// SIMATIC S7-200 project (STEP 7-Micro/WIN), CPU 224XP REL 02.01

SYMBOL_TABLE USER1
send_enable      V1020.0
gps_lat_deg      VW50
gps_lat_min      VD52
gps_lat_dir      VB56
gps_long_deg     VW57
gps_long_min     VD59
gps_long_dir     VB64
gps_alt          VD65
gps_alt_u        VB69
gps_speed        VD70
msg              VB2000
counter          VW100
counter_delay    VW102
counter_send     V10.0
counter_max      VW104
counter_stop     V10.1
table            VW2500
table_count      VW2502
table_out        VW110
table_out_s      VB112
init_pin         VB1001
init_srv         VB1006
init_busy        V1000.0
init_done        V1000.1
init_ab          V1000.2
init_st          VW1026
send_ready       V1100.3
send_to          VB1050
send_busy        V1100.0
send_done        V1100.1
send_ab          V1100.2
send_st          VW1126
send_en          V1100.4
send_stop        V1100.5
rcv_busy         V1200.0
rcv_done         V1200.1
rcv_ab           V1200.2
rcv_buf          VB1210
rcv_msg          VB1238
rcv_st           VW1250
END_SYMBOL_TABLE

ORGANIZATION_BLOCK MAIN:OB1
TITLE=PROGRAM COMMENTS
BEGIN
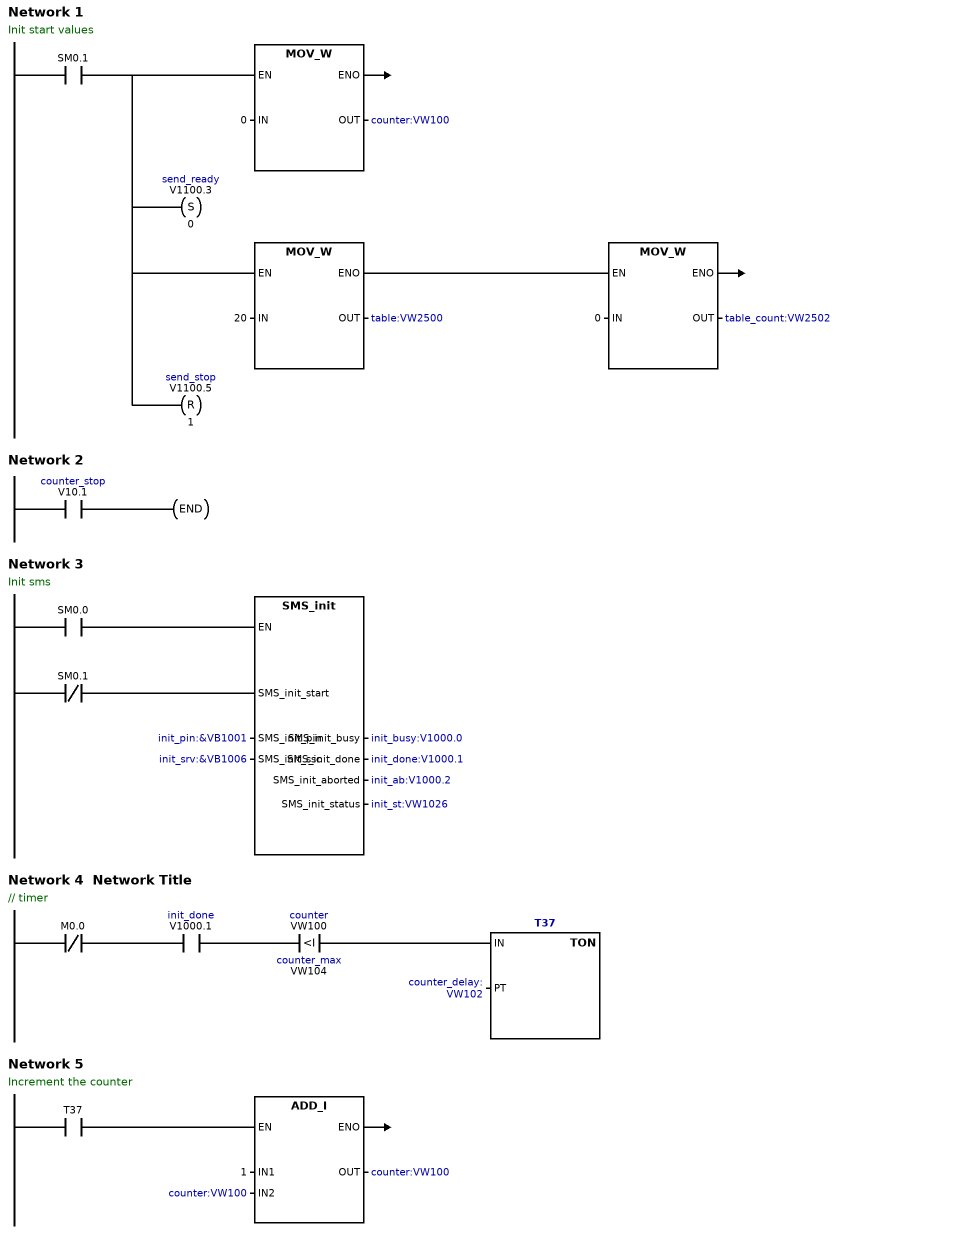
Network 1
// Init start values
LD     SM0.1
LPS
MOVW   0, counter:VW100
S      send_ready:V1100.3, 0
MOVW   20, table:VW2500
AENO
MOVW   0, table_count:VW2502
LPP
R      send_stop:V1100.5, 1
Network 2
LD     counter_stop:V10.1
END
Network 3
// Init sms
LD     SM0.0
=      L60.0
LDN    SM0.1
=      L63.7
LD     L60.0
CALL   SMS_init:SBR2, L63.7, &init_pin:VB1001, &init_srv:VB1006, init_busy:V1000.0, init_done:V1000.1, init_ab:V1000.2, init_st:VW1026
Network 4 // Network Title
// // timer
LDN    M0.0
A      init_done:V1000.1
AW<    counter:VW100, counter_max:VW104
TON    T37, counter_delay:VW102
Network 5
// Increment the counter
LD     T37
+I     1, counter:VW100
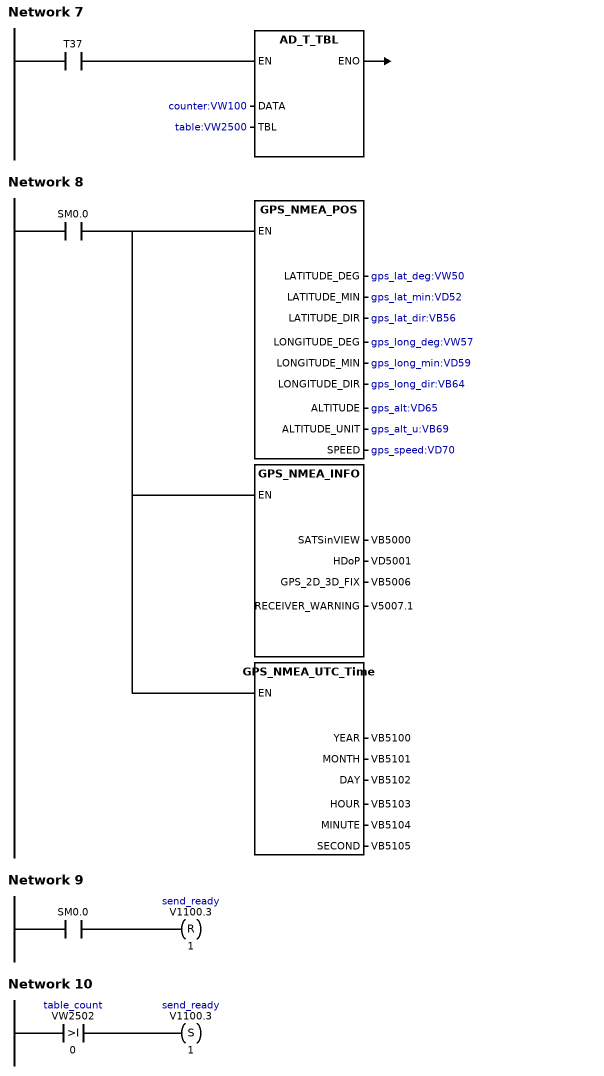
Network 7
LD     T37
ATT    counter:VW100, table:VW2500
Network 8
LD     SM0.0
CALL   GPS_NMEA_POS:SBR6, gps_lat_deg:VW50, gps_lat_min:VD52, gps_lat_dir:VB56, gps_long_deg:VW57, gps_long_min:VD59, gps_long_dir:VB64, gps_alt:VD65, gps_alt_u:VB69, gps_speed:VD70
CALL   GPS_NMEA_INFO:SBR7, VB5000, VD5001, VB5006, V5007.1
CALL   GPS_NMEA_UTC_Time:SBR8, VB5100, VB5101, VB5102, VB5103, VB5104, VB5105
Network 9
LD     SM0.0
R      send_ready:V1100.3, 1
Network 10
LDW>   table_count:VW2502, 0
S      send_ready:V1100.3, 1
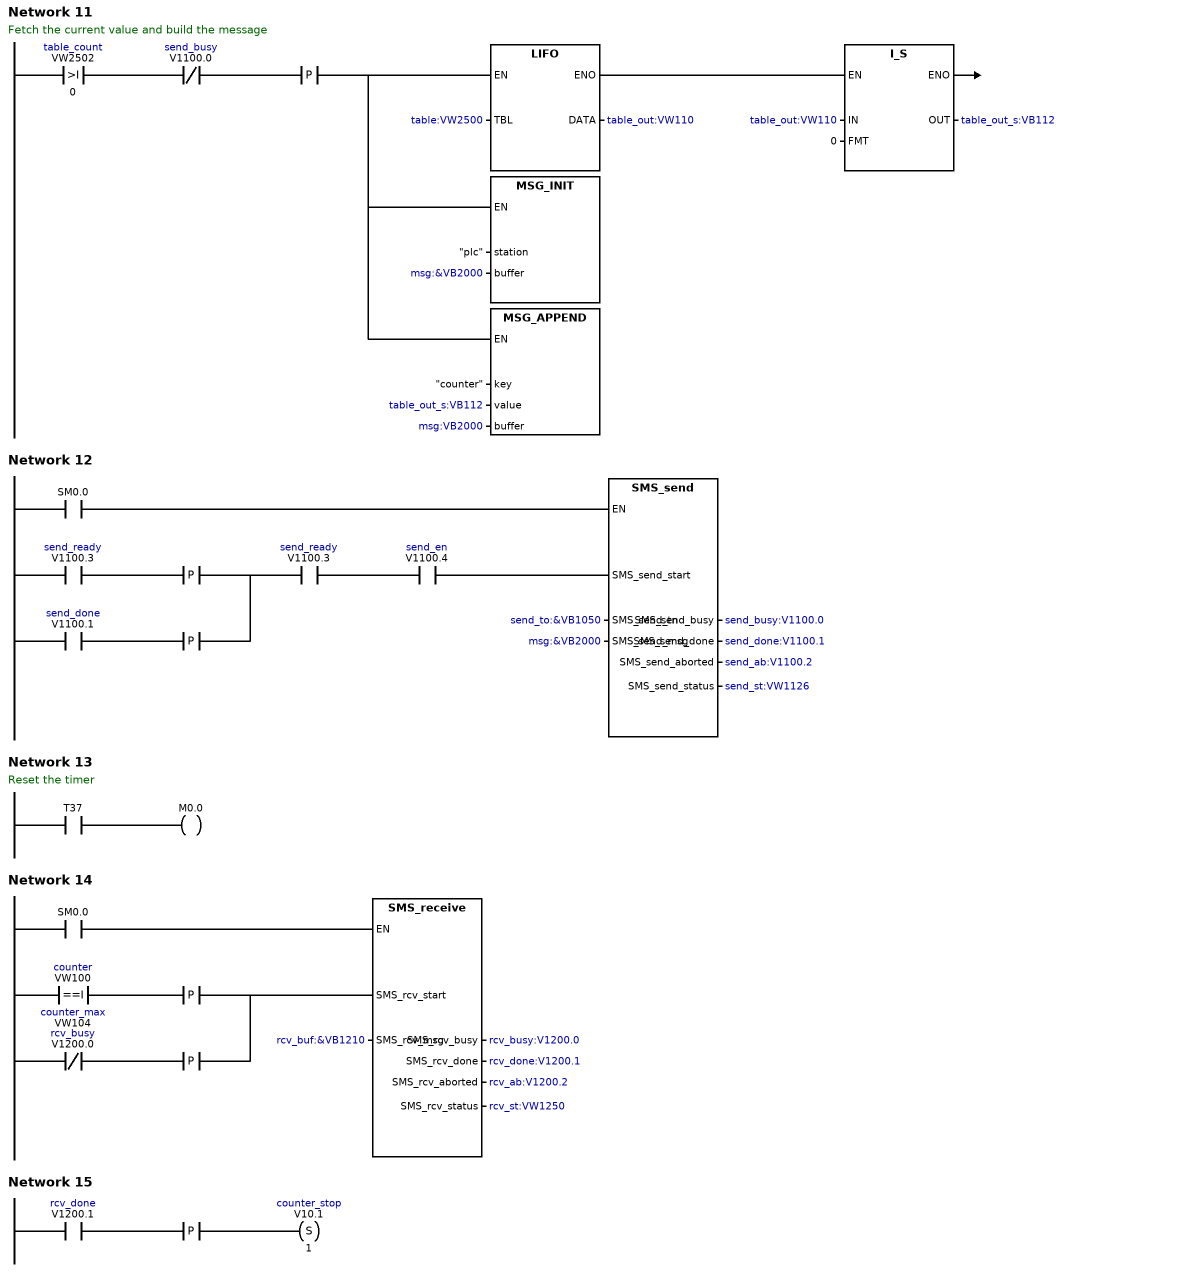
Network 11
// Fetch the current value and build the message
LDW>   table_count:VW2502, 0
AN     send_busy:V1100.0
EU
LPS
LIFO   table:VW2500, table_out:VW110
AENO
ITS    table_out:VW110, table_out_s:VB112, 0
LRD
CALL   MSG_INIT:SBR0, "plc", &msg:VB2000
LPP
CALL   MSG_APPEND:SBR5, "counter", table_out_s:VB112, msg:VB2000
Network 12
LD     SM0.0
=      L60.0
LD     send_ready:V1100.3
EU
LD     send_done:V1100.1
EU
OLD
A      send_ready:V1100.3
A      send_en:V1100.4
=      L63.7
LD     L60.0
CALL   SMS_send:SBR3, L63.7, &send_to:VB1050, &msg:VB2000, send_busy:V1100.0, send_done:V1100.1, send_ab:V1100.2, send_st:VW1126
Network 13
// Reset the timer
LD     T37
=      M0.0
Network 14
LD     SM0.0
=      L60.0
LDW=   counter:VW100, counter_max:VW104
EU
LDN    rcv_busy:V1200.0
EU
OLD
=      L63.7
LD     L60.0
CALL   SMS_receive:SBR4, L63.7, &rcv_buf:VB1210, rcv_busy:V1200.0, rcv_done:V1200.1, rcv_ab:V1200.2, rcv_st:VW1250
Network 15
LD     rcv_done:V1200.1
EU
S      counter_stop:V10.1, 1
END_ORGANIZATION_BLOCK

SUBROUTINE_BLOCK MSG_INIT:SBR0
TITLE=SUBROUTINE COMMENTS
VAR_INPUT
station:?;	// LD0 
buffer:DWORD;	// LD4 
END_VAR
VAR
year:BYTE;	// LB8 
month:BYTE;	// LB9 
day:BYTE;	// LB10 
hour:BYTE;	// LB11 
minute:BYTE;	// LB12 
seconds:BYTE;	// LB13 
tmp:INT;	// LW14 
END_VAR
BEGIN
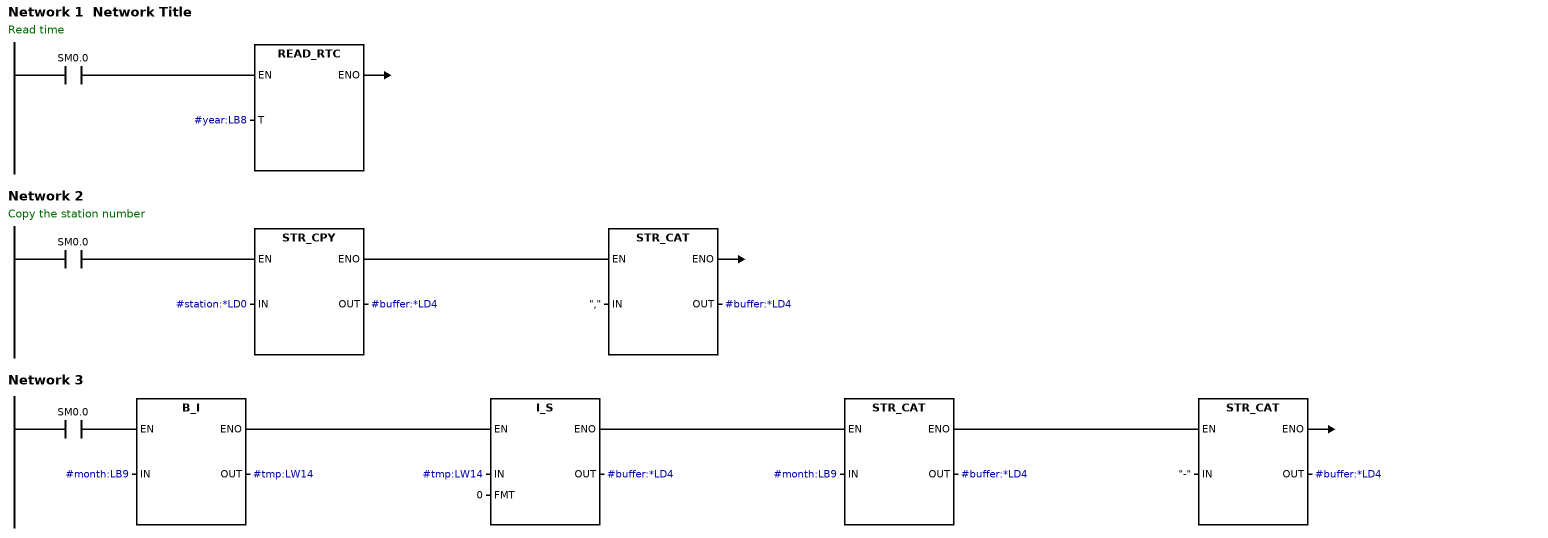
Network 1 // Network Title
// Read time
LD     SM0.0
TODR   #year:LB8
Network 2
// Copy the station number
LD     SM0.0
SCPY   *#station:LD0, *#buffer:LD4
AENO
SCAT   ",", *#buffer:LD4
Network 3
// (network saved uncompiled; LAD cells follow)
// row 0: c0 -| |- SM0.0  c1 [B_I EN:=power@row0, IN:=#month:LB9, ENO=>power, OUT=>#tmp:LW14]  c2 --  c3 --  c4 [I_S EN:=power@row0, IN:=#tmp:LW14, FMT:=0, ENO=>power, OUT=>*#buffer:LD4]  c5 --  c6 --  c7 [STR_CAT EN:=power@row0, IN:=#month:LB9, ENO=>power, OUT=>*#buffer:LD4]  c8 --  c9 --  c10 [STR_CAT EN:=power@row0, IN:="-", ENO=>power, OUT=>*#buffer:LD4]  c11 ->
// row 1: c1 [box]  c4 [box]  c7 [box]  c10 [box]
END_SUBROUTINE_BLOCK

// SBR1: protected block, not included

// SBR2: protected block, not included

// SBR3: protected block, not included

// SBR4: protected block, not included

SUBROUTINE_BLOCK MSG_APPEND:SBR5
TITLE=SUBROUTINE COMMENTS
VAR_INPUT
key:?;	// LD0 
value:?;	// LD4 
buffer:?;	// LD8 
END_VAR
BEGIN
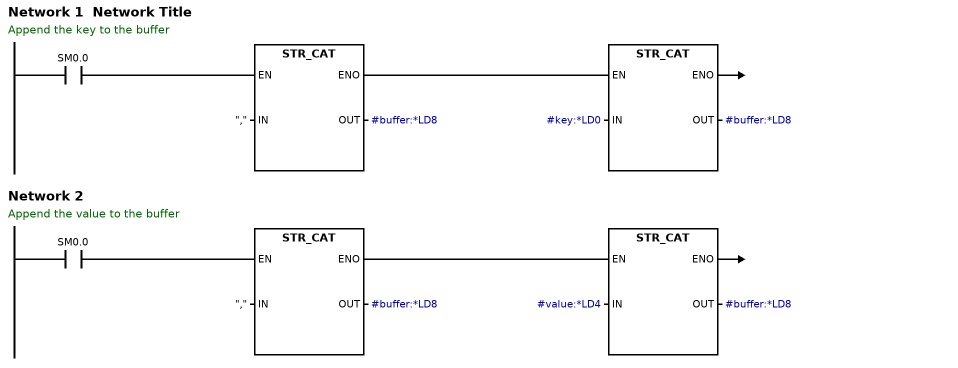
Network 1 // Network Title
// Append the key to the buffer
LD     SM0.0
SCAT   ",", *#buffer:LD8
AENO
SCAT   *#key:LD0, *#buffer:LD8
Network 2
// Append the value to the buffer
LD     SM0.0
SCAT   ",", *#buffer:LD8
AENO
SCAT   *#value:LD4, *#buffer:LD8
END_SUBROUTINE_BLOCK

// SBR6: protected block, not included

// SBR7: protected block, not included

DATA_BLOCK_TAB USER1
BEGIN
//DATA PAGE COMMENTS
//Press F1 for help and example data page
         counter_delay, 40   // counter incrementation delay, s/10
         counter_max, 3      // maximumum counter value
//table:VW2000 +20                   // counter table length
         init_pin, ""
         init_srv, "+37129202020"
         send_to, "+37129252613"
VB1100   2#0                 // enables/disables SMS sending
END_DATA_BLOCK_TAB
